(* PLC project Unnamed, Unknown Unnamed 1 *)
(* stored: creationDateTime 2023-03-10T10:37:17, modificationDateTime 2023-03-15T15:56:42 *)

(* 978-3-658-06643-7, Abb. 2.7 *)
FUNCTION_BLOCK Cylinder_Control_System
  VAR_INPUT
    INa1 : BOOL;
    INa0 : BOOL;
    INS : BOOL;
    INb1 : BOOL;
    INc0 : BOOL;
    INc1 : BOOL;
    INb0 : BOOL;
  END_VAR
  VAR_OUTPUT
    OUTBp : BOOL;
    OUTAp : BOOL;
    OUTAm : BOOL;
    OUTCp : BOOL;
  END_VAR
  VAR
    ME1 : BOOL;
    ME2 : BOOL;
  END_VAR
  VAR  (* added by the conversion: wires and edge detectors of the diagram *)
    _AND22_OUT : BOOL;
    _AND12_OUT : BOOL;
  END_VAR

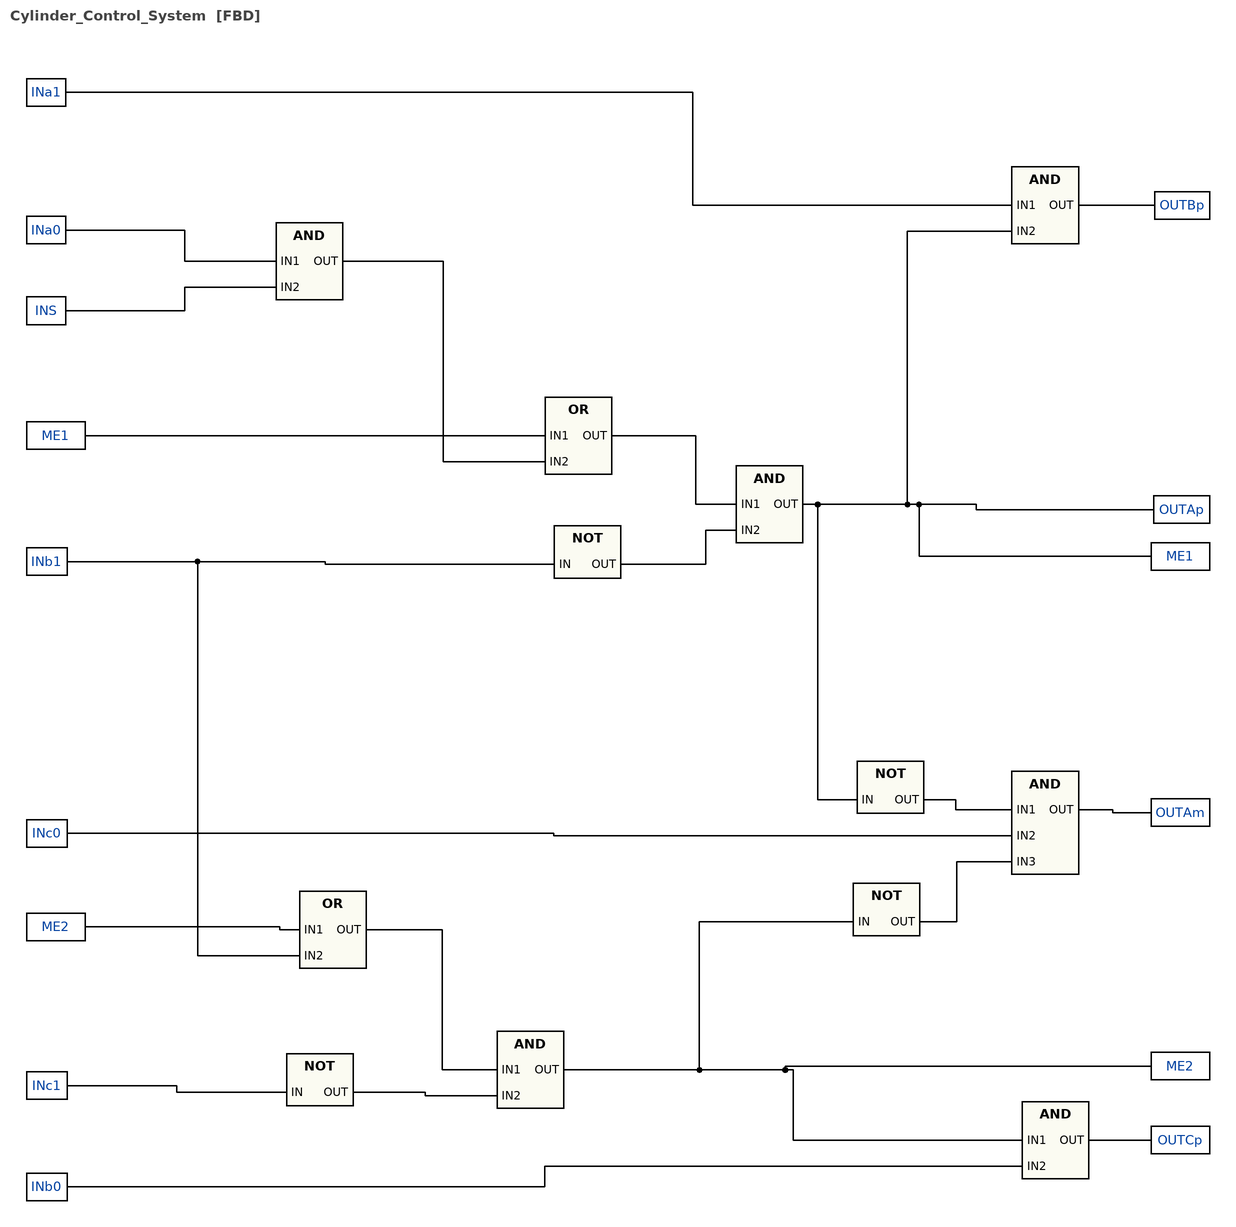
(* FBD diagram, written out as Structured Text *)
_AND22_OUT := (ME1 OR INa0 AND INS) AND NOT INb1;
OUTBp := INa1 AND _AND22_OUT;
OUTAp := _AND22_OUT;
ME1 := _AND22_OUT;
_AND12_OUT := (ME2 OR INb1) AND NOT INc1;
OUTAm := NOT _AND22_OUT AND INc0 AND NOT _AND12_OUT;
ME2 := _AND12_OUT;
OUTCp := _AND12_OUT AND INb0;
END_FUNCTION_BLOCK

CONFIGURATION config
  RESOURCE resource1 ON PLC
  END_RESOURCE
END_CONFIGURATION
